TYPE ST_MachinePondErrors_OLD :
STRUCT
	Hydraulic							: ST_HydraulicErrors;
	FeedingPulp							: ST_CilinderErrors;
	Drain								: ST_CilinderErrors;
END_STRUCT
END_TYPE

(* stored: Version 1.1.0.1, ProductVersion 3.1.4020.12
   DUT ST_MachinePondErrors_OLD: Id {856d5c73-2f85-47d0-a643-131d67f09c9d} *)
